(* IEC 61131-3 sources: PID/Source/IMM/ieccontrol/Ejector1, 4 files *)

(* ---- FBInsteadIOConfig.pu ---- *)
FUNCTION_BLOCK FBInsteadIOConfig #DUMMY_EDIT_BLOCK

VAR_INPUT
 IOPath : STRING(255);
END_VAR

VAR
 SystemPath : STRING(255) := '/harddisk0/application/control/config/KeStudio_generated/Device1/PlcIo.cfgr';
END_VAR
#BEGIN_EDIT_BLOCK
Stable_Copy := KFILE_Copy(IOPath,SystemPath);

;#END_EDIT_BLOCK END_FUNCTION_BLOCK

#END_OF_IEC_PART

@Puma @IecEditor 6 152 @Pou 25
@@@BEG_Comment@@@

@@@END_Comment@@@

@BEG_Contents

@BEG_Func
@RT(17)FuncTreeContainer
0
@END_Func

@BEG_Const
@RT(18)ConstTreeContainer
0
@END_Const

@BEG_Export

@BEG_Kind
@FUNCTION_BLOCK @RT(17)FBInsteadIOConfig @STRUCTURED_TEXT
@RT(0) @RT(0) @RT(0)
@END_Kind

@BEG_Dcl
@RT(16)DclTreeContainer
2
@Var @RT(10)SystemPath @RT(0) @T @F @DT @RT(11)STRING(255) @RT(0) @T @T @STRING 0 @F @RT(3)255 @F
@F @F
@T
@BEG_Attrib
3 @RT(77)'/harddisk0/application/control/config/KeStudio_generated/Device1/PlcIo.cfgr' @RT(0) @RT(0)
@END_Attrib
1 0 @F @F @F @F

@Var @RT(6)IOPath @RT(0) @T @F @DT @RT(11)STRING(255) @RT(0) @T @T @STRING 0 @F @RT(3)255 @F
@F @F
@T
@BEG_Attrib
3 @RT(0) @RT(0) @RT(0)
@END_Attrib
1 1 @F @F @F @F

@END_Dcl

@END_Export

@BEG_Body
@TL(2)
Stable_Copy := KFILE_Copy(IOPath,SystemPath);

@END_Body

@END_Contents

(* ---- FBReadIOConfigFiles.pu ---- *)
IMPORT_OVER_LISTFILE
 KFILE_Status
, UsbFilesArray

END_IMPORT

FUNCTION_BLOCK FBReadIOConfigFiles #DUMMY_EDIT_BLOCK

VAR_INPUT
 PLCFiles : STRING(255) := '/harddisk0/PLCIO';
END_VAR

VAR_OUTPUT
 PathArray : UsbFilesArray;
END_VAR

VAR_TEMP
 j : DINT;
END_VAR

VAR
 Stable_Free : KFILE_Status;
 Stable_First : KFILE_Status;
 Stable_Next : KFILE_Status;
 i : LINT;
 harddisk0 : STRING(255) := '/harddisk0';
 s : STRING(255);
 s2 : STRING(255);
END_VAR

(* IecGraph-Code *)

(* init step *)
INITIAL_STEP Step1:
Action1 (P);
END_STEP

ACTION Action1: #BEGIN_EDIT_BLOCK
//Check harddisk left memory
Stable_Free :=  KFILE_VolumeFree(harddisk0,i)

;#END_EDIT_BLOCK END_ACTION (*Action1*)

(* steps *)
STEP Step4:
Action3 (P);
END_STEP

ACTION Action3: #BEGIN_EDIT_BLOCK
//get first file name in the file
Stable_First := KFILE_GetFirst(PLCFiles,s);
PathArray[1] := s;
s2 := s;
FOR j :=2 TO 10 DO
   //get other file name in the file
   Stable_Next := KFILE_GetNext(s2,s2);
   PathArray[j] := s2;
END_FOR;
//Now all file name in sv_PathArray

;#END_EDIT_BLOCK END_ACTION (*Action3*)
STEP Step2:
Action5 (N);
END_STEP

ACTION Action5: #BEGIN_EDIT_BLOCK
RETURN;

;#END_EDIT_BLOCK END_ACTION (*Action5*)

(* transitions *)
TRANSITION Trans3 (* Trans3 *) FROM Step1 TO Step4 :=  #BEGIN_EDIT_BLOCK
Stable_Free = KFILE_Status_OK
;#END_EDIT_BLOCK
END_TRANSITION

TRANSITION Trans5 (* Trans5 *) FROM Step4 TO Step2 :=  #BEGIN_EDIT_BLOCK
Stable_Next = KFILE_Status_NOTOK
;#END_EDIT_BLOCK
END_TRANSITION

TRANSITION Trans2 (* Trans2 *) FROM Step2 TO Step1 :=  #BEGIN_EDIT_BLOCK
TRUE
;#END_EDIT_BLOCK
END_TRANSITION

(* end IecGraph-Code *)
(* sfc-code *)
(* end sfc-code *)

END_FUNCTION_BLOCK

#END_OF_IEC_PART

@Puma @IecEditor 6 152 @Pou 25
@@@BEG_Comment@@@

@@@END_Comment@@@

@BEG_Contents

@BEG_Func
@RT(17)FuncTreeContainer
0
@END_Func

@BEG_Const
@RT(18)ConstTreeContainer
0
@END_Const

@BEG_Export

@BEG_Kind
@FUNCTION_BLOCK @RT(19)FBReadIOConfigFiles @SEQUENTIAL_FLOW_CHART
@RT(0) @RT(0) @RT(0)
@END_Kind

@BEG_Dcl
@RT(16)DclTreeContainer
10
@Var @RT(11)Stable_Free @RT(0) @T @T @DERIVED 0 @T @T @DT @RT(12)KFILE_Status @RT(0) @T @T @UNKNOWN 0 @F
@F @F
@T
@BEG_Attrib
3 @RT(0) @RT(0) @RT(0)
@END_Attrib
1 0 @F @F @F @F

@Var @RT(12)Stable_First @RT(0) @T @T @DERIVED 0 @T @T @DT @RT(12)KFILE_Status @RT(0) @T @T @UNKNOWN 0 @F
@F @F
@T
@BEG_Attrib
3 @RT(0) @RT(0) @RT(0)
@END_Attrib
1 0 @F @F @F @F

@Var @RT(11)Stable_Next @RT(0) @T @T @DERIVED 0 @T @T @DT @RT(12)KFILE_Status @RT(0) @T @T @UNKNOWN 0 @F
@F @F
@T
@BEG_Attrib
3 @RT(0) @RT(0) @RT(0)
@END_Attrib
1 0 @F @F @F @F

@Var @RT(1)i @RT(0) @T @F @DT @RT(4)LINT @RT(0) @T @T @BASIC 0 @F
@F @F
@T
@BEG_Attrib
3 @RT(0) @RT(0) @RT(0)
@END_Attrib
1 0 @F @F @F @F

@Var @RT(1)j @RT(0) @T @F @DT @RT(4)DINT @RT(0) @T @T @BASIC 0 @F
@F @F
@T
@BEG_Attrib
3 @RT(0) @RT(0) @RT(0)
@END_Attrib
1 4 @F @F @F @F

@Var @RT(9)harddisk0 @RT(0) @T @F @DT @RT(11)STRING(255) @RT(0) @T @T @STRING 0 @F @RT(3)255 @F
@F @F
@T
@BEG_Attrib
3 @RT(12)'/harddisk0' @RT(0) @RT(0)
@END_Attrib
1 0 @F @F @F @F

@Var @RT(8)PLCFiles @RT(0) @T @F @DT @RT(11)STRING(255) @RT(0) @T @T @STRING 0 @F @RT(3)255 @F
@F @F
@T
@BEG_Attrib
3 @RT(18)'/harddisk0/PLCIO' @RT(0) @RT(0)
@END_Attrib
1 1 @F @F @F @F

@Var @RT(9)PathArray @RT(0) @T @T @DERIVED 0 @F @RT(13)UsbFilesArray @F
@T
@BEG_Attrib
3 @RT(0) @RT(0) @RT(0)
@END_Attrib
1 3 @F @F @F @F

@Var @RT(1)s @RT(0) @T @F @DT @RT(11)STRING(255) @RT(0) @T @T @STRING 0 @F @RT(3)255 @F
@F @F
@T
@BEG_Attrib
3 @RT(0) @RT(0) @RT(0)
@END_Attrib
1 0 @F @F @F @F

@Var @RT(2)s2 @RT(0) @T @F @DT @RT(11)STRING(255) @RT(0) @T @T @STRING 0 @F @RT(3)255 @F
@F @F
@T
@BEG_Attrib
3 @RT(0) @RT(0) @RT(0)
@END_Attrib
1 0 @F @F @F @F

@END_Dcl

@END_Export

@BEG_SfcBody
2 2 2

@BEG_SfcData 2
@StepSeq @RT(4)sseq @F 1
@Loop @RT(4)loop @F 2
@StepSeq @RT(3)seq @F 5
@Step @RT(5)Step1 @F @T @F @F @RT(0) @F
@AcbCont @RT(7)unnamed @F 1
@Acb @RT(7)Action1 @F @T @RT(1)P @RT(0) @F @F @T @TL(3)
//Check harddisk left memory
Stable_Free :=  KFILE_VolumeFree(harddisk0,i)

@F

@Trans @RT(6)Trans3 @F @T @F @F @T @T @TL(2)
Stable_Free = KFILE_Status_OK

@RT(6)Trans3 @F
@Step @RT(5)Step4 @F @F @F @F @RT(0) @F
@AcbCont @RT(7)unnamed @F 1
@Acb @RT(7)Action3 @F @T @RT(1)P @RT(0) @F @F @T @TL(11)
//get first file name in the file
Stable_First := KFILE_GetFirst(PLCFiles,s);
PathArray[1] := s;
s2 := s;
FOR j :=2 TO 10 DO
   //get other file name in the file
   Stable_Next := KFILE_GetNext(s2,s2);
   PathArray[j] := s2;
END_FOR;
//Now all file name in sv_PathArray

@F

@Trans @RT(6)Trans5 @F @T @F @F @T @T @TL(2)
Stable_Next = KFILE_Status_NOTOK

@RT(6)Trans5 @F
@Step @RT(5)Step2 @F @F @F @F @RT(0) @F
@AcbCont @RT(7)unnamed @F 1
@Acb @RT(7)Action5 @F @T @RT(1)N @RT(0) @F @F @T @TL(2)
RETURN;

@F

@Trans @RT(6)Trans2 @F @T @T @T @T @T @TL(2)
TRUE

@RT(6)Trans2 @F

@END_SfcData
@SaActions 0
@SaTrans 0
@SaExits 0
@END_SfcBody

@END_Contents

(* ---- ABMeasure.pu ---- *)
IMPORT_OVER_LISTFILE
 GET_MY_FU_NAME
, KSWO_AddVariable
, WRITE_SVREAL_DIRECT
, FAddToScopeGroup
, START_PROCESS_ALGORITHM
, STOP_PROCESS_ALGORITHM
, KFILE_VolumeFree
, KFILE_GetNext
, KFILE_GetFirst
, KAPPL_LintabData
, KAPPL_MeasureMonitoring
, UsbFilesArray
//  UsbFile
, FBReadIOConfigFiles
, KSWO_Status
, ABMeasureAI
, TON
, KFILE_Status
, ABPID

END_IMPORT

ALGORITHM_BLOCK ABMeasure #DUMMY_EDIT_BLOCK

SYSTEM_VAR
 sv_rEjectorPosition : REAL;
 sv_EjectorLintab : KAPPL_LintabData;
 ai_Position : REAL;
 sv_bTransducerError : BOOL;
 sv_bDeviceReady : BOOL;
 sv_rEjectorVelocity : REAL;
 sv_EjectorMonitorMeas : KAPPL_MeasureMonitoring;
 sv_Ek : REAL;
 sv_Ek_1 : REAL;
 sv_Ek_2 : REAL;
 sv_Uk : REAL;
 sv_Ui : REAL;
 sv_Uk_1 : REAL;
 sv_Uk_2 : REAL;
 sv_Uk_3 : REAL;
 di_ButtonBwd : BOOL (* Panelbutton *);
 di_ButtonFwd : BOOL (* Panelbutton *);
 ao_pid : REAL;
 sv_PathArray : UsbFilesArray;
 // sv_PathDisplay : UsbFile;
 sv_rActOutput : INT;
 sv_rSetOutput : INT;
 sv_bStartPID : BOOL;
END_VAR

SYSTEM_OBJECT
 TaskAnalog : TASK;
 TaskSlow : TASK;
 PU_Task_7 : TASK;
 // erCopyDone : ALARM;
END_OBJECT

VAR
 t : REAL := 0.2;
 T : REAL;
 Kp : REAL := 0.05;
 Ti : REAL;
 ti : REAL := 0.05;
 Td : REAL;
 td : REAL := 2.0;
 A : REAL;
 B : REAL;
 C : REAL;
 ai_pid : REAL := 10.0;
 PWMPeriod : TIME;
 T_PID : REAL;
 L_T : REAL;
 H_T : REAL;
 DutyRatio : REAL;
 fbReadIOConfigFiles : FBReadIOConfigFiles;
END_VAR

PROCESS_ALGORITHM paInitDebugMeasurement ON TaskSlow AUTOSTART

VAR
 fuName : STRING(255);
 variableName : STRING(255);
 swoState : KSWO_Status;
 b : BOOL;
END_VAR
#BEGIN_EDIT_BLOCK
fuName := GET_MY_FU_NAME();
variableName := CONCAT(fuName,'.rPosition mm');
swoState := KSWO_AddVariable( Task := TaskAnalog,
                              Name := variableName,
                              Variable := sv_rEjectorPosition);
b := FAddToScopeGroup(Task := TaskAnalog,
                      Name := variableName,
                      GroupId := cScopeGroupEjector);
variableName := CONCAT(fuName,'.rVelocity mm/s');
swoState := KSWO_AddVariable( Task := TaskAnalog,
                              Name := variableName,
                              Variable := sv_rEjectorVelocity);
b := FAddToScopeGroup(Task := TaskAnalog,
                      Name := variableName,
                      GroupId := cScopeGroupEjector);

    variableName := CONCAT(fuName,'.sv_Ek');
swoState := KSWO_AddVariable( Task := TaskAnalog,
                              Name := variableName,
                              Variable := sv_Ek);

    variableName := CONCAT(fuName,'.sv_Uk');
swoState := KSWO_AddVariable( Task := TaskAnalog,
                              Name := variableName,
                              Variable := sv_Uk);

    variableName := CONCAT(fuName,'.sv_Ui');
swoState := KSWO_AddVariable( Task := TaskAnalog,
                              Name := variableName,
                              Variable := sv_Ui);

    variableName := CONCAT(fuName,'.ao_pid');
swoState := KSWO_AddVariable( Task := TaskAnalog,
                              Name := variableName,
                              Variable := ao_pid);

    variableName := CONCAT(fuName,'.ai_pid');
swoState := KSWO_AddVariable( Task := TaskAnalog,
                              Name := variableName,
                              Variable := ai_pid);

    variableName := CONCAT(fuName,'.sv_rActOutput');
swoState := KSWO_AddVariable( Task := TaskAnalog,
                              Name := variableName,
                              Variable := sv_rActOutput);
    variableName := CONCAT(fuName,'.sv_rSetOutput');
swoState := KSWO_AddVariable( Task := TaskAnalog,
                              Name := variableName,
                              Variable := sv_rSetOutput);

STOP_PROCESS_ALGORITHM();

;#END_EDIT_BLOCK END_ALGORITHM

PROCESS_ALGORITHM paMeasure ON TaskAnalog AUTOSTART

VAR_TEMP
 b : BOOL;
END_VAR

VAR
 abEjectorMeasure : ABMeasureAI;
END_VAR

(* IecGraph-Code *)

(* init step *)
INITIAL_STEP S_Start:
END_STEP

(* steps *)
STEP S_Stop:
AStop (P);
END_STEP

ACTION AStop: #BEGIN_EDIT_BLOCK
STOP_PROCESS_ALGORITHM();

;#END_EDIT_BLOCK END_ACTION (*AStop*)
STEP S_Init:
AInitMeasureBlock (P);
END_STEP

STEP S_Measure:
AMeasure (N);
END_STEP

(* transitions *)
TRANSITION TLinked (* TLinked *) FROM S_Start TO S_Init :=  #BEGIN_EDIT_BLOCK
IS_LINKED(ai_Position)
;#END_EDIT_BLOCK
END_TRANSITION

TRANSITION TNotLinked (* TNotLinked *) FROM S_Start TO S_Stop :=  #BEGIN_EDIT_BLOCK
NOT IS_LINKED(ai_Position)
;#END_EDIT_BLOCK
END_TRANSITION

TRANSITION TStop (* TStop *) FROM S_Stop TO S_Start :=  #BEGIN_EDIT_BLOCK
TRUE
;#END_EDIT_BLOCK
END_TRANSITION

TRANSITION TInitDone (* TInitDone *) FROM S_Init TO S_Measure :=  #BEGIN_EDIT_BLOCK
TRUE
;#END_EDIT_BLOCK
END_TRANSITION

(* end IecGraph-Code *)
(* sfc-code *)

(* stand alone actions *)
ACTION AMeasure: #BEGIN_EDIT_BLOCK

abEjectorMeasure.aRun(bIdle := sv_bDeviceReady);
sv_bTransducerError := abEjectorMeasure.aRun.bSensorError;
b := WRITE_SVREAL_DIRECT(sv_rEjectorPosition, abEjectorMeasure.aRun.rValue);
b := WRITE_SVREAL_DIRECT(sv_rEjectorVelocity, abEjectorMeasure.aRun.rVelocity);

;#END_EDIT_BLOCK END_ACTION (*AMeasure*)
ACTION AInitMeasureBlock: #BEGIN_EDIT_BLOCK

abEjectorMeasure.aInit(sRawValue := 'Ejector1.ai_Position',
                        pLintab := @sv_EjectorLintab);

abEjectorMeasure.aInitMonitoring(bEnable := sv_EjectorMonitorMeas.EnableMonitoring,
                                 rLowLimit := sv_EjectorMonitorMeas.LowerLimit,
                                 bLimitation := sv_EjectorMonitorMeas.Limitation,
                                 rFailureFactor := sv_EjectorMonitorMeas.FailureFactor);

;#END_EDIT_BLOCK END_ACTION (*AInitMeasureBlock*)
(* end sfc-code *)

END_ALGORITHM

PROCESS_ALGORITHM paPID ON TaskAnalog

(* IecGraph-Code *)

(* init step *)
INITIAL_STEP Step1:
Action223 (P);
END_STEP

ACTION Action223: #BEGIN_EDIT_BLOCK
ai_pid := 10.0;
t := 0.1;
td := 2.0;
ti := 0.05;
Kp := 0.2;

;#END_EDIT_BLOCK END_ACTION (*Action223*)

(* steps *)
STEP Step2:
Action2 (P);
END_STEP

ACTION Action2: #BEGIN_EDIT_BLOCK
sv_Ek := 0.0;
sv_Ek_1 := 0.0;
sv_Ek_2 := 0.0;
sv_Uk := 0.0;
sv_Uk_1 := 0.0;
sv_Uk_2 := 0.0;
sv_Uk_3 := 0.0;

;#END_EDIT_BLOCK END_ACTION (*Action2*)
STEP Step4:
END_STEP

STEP Step3:
Action3 (P);
END_STEP

ACTION Action3: #BEGIN_EDIT_BLOCK
T := 1.0/t;
Td := 1.0/td;
Ti := 1.0/ti;
A := Kp*(1.0 + T/Ti + Td/T);
B := Kp*(1.0 + 2.0*Td/T);
C := Kp*Td/T;
sv_Uk_3 := sv_Uk_2;
sv_Uk_2 := sv_Uk_1;
sv_Uk_1 := sv_Uk;
sv_Ek_2 := sv_Ek_1;
sv_Ek_1 := sv_Ek;
sv_Ek := ai_pid - sv_Uk;
sv_Ui := A*sv_Ek + B*sv_Ek_1 + C*sv_Ek_2;
ao_pid := sv_Uk_1 + sv_Ui;
sv_Uk := sv_Uk_1 + sv_Ui;

;#END_EDIT_BLOCK END_ACTION (*Action3*)

(* transitions *)
GO_ON_TRANSITION Trans1 (* Trans1 *) FROM Step1 TO Step2 :=  #BEGIN_EDIT_BLOCK
TRUE
;#END_EDIT_BLOCK
END_TRANSITION

TRANSITION Trans4 (* Trans4 *) FROM Step2 TO Step4 :=  #BEGIN_EDIT_BLOCK
TRUE
;#END_EDIT_BLOCK
END_TRANSITION

TRANSITION Trans2 (* Trans2 *) FROM Step4 TO Step3 :=  #BEGIN_EDIT_BLOCK
Step4.T > t#0.1s
;#END_EDIT_BLOCK
END_TRANSITION

GO_ON_TRANSITION Trans5 (* Trans5 *) FROM Step3 TO Step4 :=  #BEGIN_EDIT_BLOCK
TRUE
;#END_EDIT_BLOCK
END_TRANSITION

(* end IecGraph-Code *)
(* sfc-code *)
(* end sfc-code *)

END_ALGORITHM

POSTUPDATE_ALGORITHM p ON PU_Task_7 WITH di_ButtonBwd,di_ButtonFwd

VAR
 a : INT;
END_VAR
#BEGIN_EDIT_BLOCK

IF di_ButtonFwd THEN
   START_PROCESS_ALGORITHM(paPID);
   START_PROCESS_ALGORITHM(paPWM);

END_IF;

IF di_ButtonBwd THEN
   STOP_PROCESS_ALGORITHM(paPID);
   STOP_PROCESS_ALGORITHM(paPWM);
END_IF;
//year=(year%100==0)?(year%400==0?1:0):(year%4==0?1:0)

;#END_EDIT_BLOCK END_ALGORITHM

PROCESS_ALGORITHM paPWM ON TaskAnalog

VAR
 fbTON : TON;
 do : BOOL;
END_VAR

(* IecGraph-Code *)

(* init step *)
INITIAL_STEP Step1:
Action20 (P);
END_STEP

ACTION Action20: #BEGIN_EDIT_BLOCK
PWMPeriod := t#2s;

;#END_EDIT_BLOCK END_ACTION (*Action20*)

(* steps *)
STEP Step2:
Action2 (P);
END_STEP

ACTION Action2: #BEGIN_EDIT_BLOCK
T_PID := ao_pid;
L_T := 8.0;
H_T := 10.0;
IF T_PID < L_T THEN
   DutyRatio := 1.0;
ELSE IF T_PID >= H_T - 0.1 THEN
   DutyRatio := 0.0;
ELSE
   DutyRatio := (T_PID - L_T) /(H_T - L_T);
END_IF;
END_IF;
fbTON(IN := FALSE);

;#END_EDIT_BLOCK END_ACTION (*Action2*)
STEP Step5:
Action3 (N);
END_STEP

ACTION Action3: #BEGIN_EDIT_BLOCK
fbTON(IN := TRUE,
     // PT := REAL_TO_TIME(TIME_TO_REAL(PWMPeriod) * DutyRatio);
            PT := PWMPeriod * DutyRatio);
IF fbTON.Q THEN
   do := FALSE;
ELSE
   do := TRUE;
END_IF;

;#END_EDIT_BLOCK END_ACTION (*Action3*)
STEP Step3:
END_STEP

(* transitions *)
TRANSITION Trans1 (* Trans1 *) FROM Step1 TO Step2 :=  #BEGIN_EDIT_BLOCK
TRUE
;#END_EDIT_BLOCK
END_TRANSITION

TRANSITION Trans2 (* Trans2 *) FROM Step2 TO Step5 :=  #BEGIN_EDIT_BLOCK
TRUE
;#END_EDIT_BLOCK
END_TRANSITION

TRANSITION Trans11 (* Trans11 *) FROM Step5 TO Step3 :=  #BEGIN_EDIT_BLOCK
Step5.T > PWMPeriod
;#END_EDIT_BLOCK
END_TRANSITION

TRANSITION Trans12 (* Trans12 *) FROM Step3 TO Step2 :=  #BEGIN_EDIT_BLOCK
TRUE
;#END_EDIT_BLOCK
END_TRANSITION

(* end IecGraph-Code *)
(* sfc-code *)
(* end sfc-code *)

END_ALGORITHM

POSTUPDATE_ALGORITHM USB ON PU_Task_7 WITH di_ButtonBwd,di_ButtonFwd

VAR
 PLCFiles : STRING(255) := '/harddisk0/PLCIO';
END_VAR
#BEGIN_EDIT_BLOCK
IF di_ButtonBwd THEN
   START_PROCESS_ALGORITHM(paUSB);
END_IF;
IF di_ButtonFwd THEN
   STOP_PROCESS_ALGORITHM(paUSB);
END_IF;

;#END_EDIT_BLOCK END_ALGORITHM

PROCESS_ALGORITHM paUSB ON TaskAnalog

VAR_TEMP
 j : DINT;
END_VAR

VAR
 Stable_Free : KFILE_Status;
 Stable_Delete : KFILE_Status;
 Stable_Copy : KFILE_Status;
 Stable_Next : KFILE_Status;
 Stable_First : KFILE_Status;
 Stable_Copy2 : KFILE_Status;
 Stable_Rename : KFILE_Status;
 i : LINT;
 SystemPath : STRING(255) := '/harddisk0/application/control/config/KeStudio_generated/Device1/PlcIo.cfgr';
 s : STRING(255);
 s2 : STRING(255);
 harddisk0 : STRING(255) := '/harddisk0';
 PLCFiles : STRING(255) := '/harddisk0';
END_VAR

(* IecGraph-Code *)

(* init step *)
INITIAL_STEP Step1:
Action1 (P);
END_STEP

ACTION Action1: #BEGIN_EDIT_BLOCK
//Check harddisk left memory
Stable_Free :=  KFILE_VolumeFree(harddisk0,i)

;#END_EDIT_BLOCK END_ACTION (*Action1*)

(* steps *)
STEP Step4:
Action3 (P);
END_STEP

ACTION Action3: #BEGIN_EDIT_BLOCK
//get first file name in the file
Stable_First := KFILE_GetFirst(PLCFiles,s);
sv_PathArray[1] := s;
s2 := s;
FOR j :=2 TO 10 DO
   //get other file name in the file
   Stable_Next := KFILE_GetNext(s2,s2);
   sv_PathArray[j] := s2;
END_FOR;
//Now all file name in sv_PathArray

;#END_EDIT_BLOCK END_ACTION (*Action3*)
STEP Step2:
Action5 (N);
END_STEP

ACTION Action5: #BEGIN_EDIT_BLOCK

STOP_PROCESS_ALGORITHM();

;#END_EDIT_BLOCK END_ACTION (*Action5*)

(* transitions *)
TRANSITION Trans3 (* Trans3 *) FROM Step1 TO Step4 :=  #BEGIN_EDIT_BLOCK
Stable_Free = KFILE_Status_OK
;#END_EDIT_BLOCK
END_TRANSITION

TRANSITION Trans5 (* Trans5 *) FROM Step4 TO Step2 :=  #BEGIN_EDIT_BLOCK
Stable_Next = KFILE_Status_NOTOK
;#END_EDIT_BLOCK
END_TRANSITION

TRANSITION Trans2 (* Trans2 *) FROM Step2 TO Step1 :=  #BEGIN_EDIT_BLOCK
TRUE
;#END_EDIT_BLOCK
END_TRANSITION

(* end IecGraph-Code *)
(* sfc-code *)
(* end sfc-code *)

END_ALGORITHM

// POSTUPDATE_ALGORITHM pchoose ON PU_Task_7 WITH sv_bUse1,sv_bUse2,sv_bUse3,sv_bUse4,sv_bUse5,sv_bUse6,sv_bUse7,sv_bUse8,sv_bUse9,sv_bUse10

// VAR
 // Stable_Copy : KFILE_Status;
 // SystemPath : STRING(255) := '/harddisk0/application/control/config/KeStudio_generated/Device1/PlcIo.cfgr';
// END_VAR
// #BEGIN_EDIT_BLOCK
// IF sv_bUse1 THEN
// Stable_Copy := KFILE_Copy(sv_PathDisplay.plc1,SystemPath);
// END_IF;
//
// IF sv_bUse2 THEN
// Stable_Copy := KFILE_Copy(sv_PathDisplay.plc2,SystemPath);
// END_IF;
//
// IF sv_bUse3  THEN
// Stable_Copy := KFILE_Copy(sv_PathDisplay.plc3,SystemPath);
// END_IF;
//
// IF sv_bUse4 THEN
// Stable_Copy := KFILE_Copy(sv_PathDisplay.plc4,SystemPath);
// END_IF;
//
// IF sv_bUse5 THEN
// Stable_Copy := KFILE_Copy(sv_PathDisplay.plc5,SystemPath);
// END_IF;
//
// IF sv_bUse6 THEN
// Stable_Copy := KFILE_Copy(sv_PathDisplay.plc6,SystemPath);
// END_IF;
//
// IF sv_bUse7 THEN
// Stable_Copy := KFILE_Copy(sv_PathDisplay.plc7,SystemPath);
// END_IF;
//
// IF sv_bUse8 THEN
// Stable_Copy := KFILE_Copy(sv_PathDisplay.plc8,SystemPath);
// END_IF;
//
// IF sv_bUse9 THEN
// Stable_Copy := KFILE_Copy(sv_PathDisplay.plc9,SystemPath);
// END_IF;
//
// IF sv_bUse10 THEN
// Stable_Copy := KFILE_Copy(sv_PathDisplay.plc10,SystemPath);
// END_IF;
//

// ;#END_EDIT_BLOCK END_ALGORITHM

// PROCESS_ALGORITHM paPIDCalc ON TaskAnalog AUTOSTART

// #BEGIN_EDIT_BLOCK
// Td := 1.0/td;
// Ti := 1.0/ti;
// A := Kp*(1.0 + T/Ti + Td/T);
// B := Kp*(1.0 + 2.0*Td/T);
// C := Kp*Td/T;
// sv_Uk_3 := sv_Uk_2;
// sv_Uk_2 := sv_Uk_1;
// sv_Uk_1 := sv_Uk;
// sv_Ek_2 := sv_Ek_1;
// sv_Ek_1 := sv_Ek;
// sv_Ek := ai_pid - sv_Uk;
// sv_Ui := A*sv_Ek + B*sv_Ek_1 + C*sv_Ek_2;
// ao_pid := sv_Uk_1 + sv_Ui;
// sv_Uk := sv_Uk_1 + sv_Ui;

// ;#END_EDIT_BLOCK END_ALGORITHM

PROCESS_ALGORITHM pStaratPID ON TaskSlow AUTOSTART

VAR
 iKp : INT := 2;
 iKd : INT := 1;
 iKi : INT := 1;
 iFilter : INT := 1023;
 iIntegr : INT := 0;
 abPID : ABPID;
END_VAR
#BEGIN_EDIT_BLOCK
IF sv_bStartPID THEN
    abPID.aPID(iAct := (sv_rActOutput * 32/ 100),
         iSet := (sv_rSetOutput * 32 / 100),
         iKp := iKp,
         iKi := iKi,
         iKd := iKd,
         iC0 := iFilter,
         iYlow := -32,
         iYup := 32,
         iIntegr := iIntegr,
         iY => sv_rActOutput);
   iIntegr := abPID.aPID.iIntegr;

END_IF;

;#END_EDIT_BLOCK END_ALGORITHM

END_ALGORITHM_BLOCK

#END_OF_IEC_PART

@Puma @IecEditor 6 103 @Pou 25
@@@BEG_Comment@@@

@@@END_Comment@@@

@BEG_Contents

@BEG_Func
@RT(17)FuncTreeContainer
9
@Var @RT(14)GET_MY_FU_NAME @RT(0) @T @T @DERIVED 0 @F @RT(22)KEBA_STANDARD_FUNCTION @F
@T
@BEG_Attrib
0 @RT(0) @RT(0)
@END_Attrib
1 1 @F @F @F @F

@Var @RT(16)KSWO_AddVariable @RT(0) @T @T @DERIVED 0 @F @RT(22)KEBA_STANDARD_FUNCTION @F
@T
@BEG_Attrib
0 @RT(0) @RT(0)
@END_Attrib
1 1 @F @F @F @F

@Var @RT(19)WRITE_SVREAL_DIRECT @RT(0) @T @T @DERIVED 0 @F @RT(22)KEBA_STANDARD_FUNCTION @F
@T
@BEG_Attrib
0 @RT(0) @RT(0)
@END_Attrib
1 1 @F @F @F @F

@Var @RT(16)FAddToScopeGroup @RT(0) @T @T @DERIVED 0 @F @RT(8)FUNCTION @F
@T
@BEG_Attrib
0 @RT(0) @RT(0)
@END_Attrib
1 1 @F @F @F @F

@Var @RT(23)START_PROCESS_ALGORITHM @RT(0) @T @T @DERIVED 0 @F @RT(23)KEBA_STANDARD_PROCEDURE @F
@T
@BEG_Attrib
0 @RT(0) @RT(0)
@END_Attrib
1 1 @F @F @F @F

@Var @RT(22)STOP_PROCESS_ALGORITHM @RT(0) @T @T @DERIVED 0 @F @RT(23)KEBA_STANDARD_PROCEDURE @F
@T
@BEG_Attrib
0 @RT(0) @RT(0)
@END_Attrib
1 1 @F @F @F @F

@Var @RT(16)KFILE_VolumeFree @RT(0) @T @T @DERIVED 0 @F @RT(22)KEBA_STANDARD_FUNCTION @F
@T
@BEG_Attrib
0 @RT(0) @RT(0)
@END_Attrib
1 1 @F @F @F @F

@Var @RT(13)KFILE_GetNext @RT(0) @T @T @DERIVED 0 @F @RT(22)KEBA_STANDARD_FUNCTION @F
@T
@BEG_Attrib
0 @RT(0) @RT(0)
@END_Attrib
1 1 @F @F @F @F

@Var @RT(14)KFILE_GetFirst @RT(0) @T @T @DERIVED 0 @F @RT(22)KEBA_STANDARD_FUNCTION @F
@T
@BEG_Attrib
0 @RT(0) @RT(0)
@END_Attrib
1 1 @F @F @F @F

@END_Func

@BEG_Const
@RT(18)ConstTreeContainer
0
@END_Const

@BEG_Export

@BEG_Kind
@ALGORITHM_BLOCK @RT(9)ABMeasure @STRUCTURED_TEXT
@RT(0) @RT(0) @RT(0)
@END_Kind

@BEG_Dcl
@RT(16)DclTreeContainer
44
@Var @RT(19)sv_rEjectorPosition @RT(0) @T @F @DT @RT(4)REAL @RT(0) @T @T @BASIC 0 @F
@F @F
@T
@BEG_Attrib
3 @RT(0) @RT(0) @RT(0)
@END_Attrib
1 8 @F @F @F @F

@Var @RT(16)sv_EjectorLintab @RT(0) @T @T @DERIVED 0 @T @T @DT @RT(16)KAPPL_LintabData @RT(0) @T @T @UNKNOWN 0 @F
@F @F
@T
@BEG_Attrib
3 @RT(0) @RT(0) @RT(0)
@END_Attrib
1 8 @F @F @F @F

@Var @RT(11)ai_Position @RT(0) @T @F @DT @RT(4)REAL @RT(0) @T @T @BASIC 0 @F
@F @F
@T
@BEG_Attrib
3 @RT(0) @RT(0) @RT(0)
@END_Attrib
1 8 @F @F @F @F

@Var @RT(19)sv_bTransducerError @RT(0) @T @F @DT @RT(4)BOOL @RT(0) @T @T @BASIC 0 @F
@F @F
@T
@BEG_Attrib
3 @RT(0) @RT(0) @RT(0)
@END_Attrib
1 8 @F @F @F @F

@Var @RT(15)sv_bDeviceReady @RT(0) @T @F @DT @RT(4)BOOL @RT(0) @T @T @BASIC 0 @F
@F @F
@T
@BEG_Attrib
3 @RT(0) @RT(0) @RT(0)
@END_Attrib
1 8 @F @F @F @F

@Var @RT(19)sv_rEjectorVelocity @RT(0) @T @F @DT @RT(4)REAL @RT(0) @T @T @BASIC 0 @F
@F @F
@T
@BEG_Attrib
3 @RT(0) @RT(0) @RT(0)
@END_Attrib
1 8 @F @F @F @F

@Var @RT(21)sv_EjectorMonitorMeas @RT(0) @T @T @DERIVED 0 @T @T @DT @RT(23)KAPPL_MeasureMonitoring @RT(0) @T @T @UNKNOWN 0 @F
@F @F
@T
@BEG_Attrib
3 @RT(0) @RT(0) @RT(0)
@END_Attrib
1 8 @F @F @F @F

@Var @RT(10)TaskAnalog @RT(0) @T @F @DT @RT(4)TASK @RT(0) @T @T @BASIC 0 @F
@F @F
@T
@BEG_Attrib
3 @RT(0) @RT(0) @RT(0)
@END_Attrib
1 7 @F @F @F @F

@Var @RT(8)TaskSlow @RT(0) @T @F @DT @RT(4)TASK @RT(0) @T @T @BASIC 0 @F
@F @F
@T
@BEG_Attrib
3 @RT(0) @RT(0) @RT(0)
@END_Attrib
1 7 @F @F @F @F

@Var @RT(5)sv_Ek @RT(0) @T @F @DT @RT(4)REAL @RT(0) @T @T @BASIC 0 @F
@F @F
@T
@BEG_Attrib
3 @RT(0) @RT(0) @RT(0)
@END_Attrib
1 8 @F @F @F @F

@Var @RT(7)sv_Ek_1 @RT(0) @T @F @DT @RT(4)REAL @RT(0) @T @T @BASIC 0 @F
@F @F
@T
@BEG_Attrib
3 @RT(0) @RT(0) @RT(0)
@END_Attrib
1 8 @F @F @F @F

@Var @RT(7)sv_Ek_2 @RT(0) @T @F @DT @RT(4)REAL @RT(0) @T @T @BASIC 0 @F
@F @F
@T
@BEG_Attrib
3 @RT(0) @RT(0) @RT(0)
@END_Attrib
1 8 @F @F @F @F

@Var @RT(5)sv_Uk @RT(0) @T @F @DT @RT(4)REAL @RT(0) @T @T @BASIC 0 @F
@F @F
@T
@BEG_Attrib
3 @RT(0) @RT(0) @RT(0)
@END_Attrib
1 8 @F @F @F @F

@Var @RT(5)sv_Ui @RT(0) @T @F @DT @RT(4)REAL @RT(0) @T @T @BASIC 0 @F
@F @F
@T
@BEG_Attrib
3 @RT(0) @RT(0) @RT(0)
@END_Attrib
1 8 @F @F @F @F

@Var @RT(7)sv_Uk_1 @RT(0) @T @F @DT @RT(4)REAL @RT(0) @T @T @BASIC 0 @F
@F @F
@T
@BEG_Attrib
3 @RT(0) @RT(0) @RT(0)
@END_Attrib
1 8 @F @F @F @F

@Var @RT(7)sv_Uk_2 @RT(0) @T @F @DT @RT(4)REAL @RT(0) @T @T @BASIC 0 @F
@F @F
@T
@BEG_Attrib
3 @RT(0) @RT(0) @RT(0)
@END_Attrib
1 8 @F @F @F @F

@Var @RT(7)sv_Uk_3 @RT(0) @T @F @DT @RT(4)REAL @RT(0) @T @T @BASIC 0 @F
@F @F
@T
@BEG_Attrib
3 @RT(0) @RT(0) @RT(0)
@END_Attrib
1 8 @F @F @F @F

@Var @RT(1)t @RT(0) @T @F @DT @RT(4)REAL @RT(0) @T @T @BASIC 0 @F
@F @F
@T
@BEG_Attrib
3 @RT(3)0.2 @RT(0) @RT(0)
@END_Attrib
1 0 @F @F @F @F

@Var @RT(1)T @RT(0) @T @F @DT @RT(4)REAL @RT(0) @T @T @BASIC 0 @F
@F @F
@T
@BEG_Attrib
3 @RT(0) @RT(0) @RT(0)
@END_Attrib
1 0 @F @F @F @F

@Var @RT(2)Kp @RT(0) @T @F @DT @RT(4)REAL @RT(0) @T @T @BASIC 0 @F
@F @F
@T
@BEG_Attrib
3 @RT(4)0.05 @RT(0) @RT(0)
@END_Attrib
1 0 @F @F @F @F

@Var @RT(2)Ti @RT(0) @T @F @DT @RT(4)REAL @RT(0) @T @T @BASIC 0 @F
@F @F
@T
@BEG_Attrib
3 @RT(0) @RT(0) @RT(0)
@END_Attrib
1 0 @F @F @F @F

@Var @RT(2)ti @RT(0) @T @F @DT @RT(4)REAL @RT(0) @T @T @BASIC 0 @F
@F @F
@T
@BEG_Attrib
3 @RT(4)0.05 @RT(0) @RT(0)
@END_Attrib
1 0 @F @F @F @F

@Var @RT(2)Td @RT(0) @T @F @DT @RT(4)REAL @RT(0) @T @T @BASIC 0 @F
@F @F
@T
@BEG_Attrib
3 @RT(0) @RT(0) @RT(0)
@END_Attrib
1 0 @F @F @F @F

@Var @RT(2)td @RT(0) @T @F @DT @RT(4)REAL @RT(0) @T @T @BASIC 0 @F
@F @F
@T
@BEG_Attrib
3 @RT(3)2.0 @RT(0) @RT(0)
@END_Attrib
1 0 @F @F @F @F

@Var @RT(1)A @RT(0) @T @F @DT @RT(4)REAL @RT(0) @T @T @BASIC 0 @F
@F @F
@T
@BEG_Attrib
3 @RT(0) @RT(0) @RT(0)
@END_Attrib
1 0 @F @F @F @F

@Var @RT(1)B @RT(0) @T @F @DT @RT(4)REAL @RT(0) @T @T @BASIC 0 @F
@F @F
@T
@BEG_Attrib
3 @RT(0) @RT(0) @RT(0)
@END_Attrib
1 0 @F @F @F @F

@Var @RT(1)C @RT(0) @T @F @DT @RT(4)REAL @RT(0) @T @T @BASIC 0 @F
@F @F
@T
@BEG_Attrib
3 @RT(0) @RT(0) @RT(0)
@END_Attrib
1 0 @F @F @F @F

@Var @RT(12)di_ButtonBwd @RT(0) @T @F @DT @RT(4)BOOL @RT(0) @T @T @BASIC 0 @F
@F @F
@T
@BEG_Attrib
3 @RT(0) @RT(11)Panelbutton @RT(0)
@END_Attrib
1 8 @F @F @F @F

@Var @RT(12)di_ButtonFwd @RT(0) @T @F @DT @RT(4)BOOL @RT(0) @T @T @BASIC 0 @F
@F @F
@T
@BEG_Attrib
3 @RT(0) @RT(11)Panelbutton @RT(0)
@END_Attrib
1 8 @F @F @F @F

@Var @RT(6)ao_pid @RT(0) @T @F @DT @RT(4)REAL @RT(0) @T @T @BASIC 0 @F
@F @F
@T
@BEG_Attrib
3 @RT(0) @RT(0) @RT(0)
@END_Attrib
1 8 @F @F @F @F

@Var @RT(6)ai_pid @RT(0) @T @F @DT @RT(4)REAL @RT(0) @T @T @BASIC 0 @F
@F @F
@T
@BEG_Attrib
3 @RT(4)10.0 @RT(0) @RT(0)
@END_Attrib
1 0 @F @F @F @F

@Var @RT(9)PU_Task_7 @RT(0) @T @T @RENAMED 0 @T @T @DT @RT(4)TASK @RT(0) @T @T @BASIC 0 @F
@F @F
@T
@BEG_Attrib
3 @RT(0) @RT(0) @RT(0)
@END_Attrib
1 7 @F @F @F @F

@Var @RT(9)PWMPeriod @RT(0) @T @F @DT @RT(4)TIME @RT(0) @T @T @BASIC 0 @F
@F @F
@T
@BEG_Attrib
3 @RT(0) @RT(0) @RT(0)
@END_Attrib
1 0 @F @F @F @F

@Var @RT(5)T_PID @RT(0) @T @F @DT @RT(4)REAL @RT(0) @T @T @BASIC 0 @F
@F @F
@T
@BEG_Attrib
3 @RT(0) @RT(0) @RT(0)
@END_Attrib
1 0 @F @F @F @F

@Var @RT(3)L_T @RT(0) @T @F @DT @RT(4)REAL @RT(0) @T @T @BASIC 0 @F
@F @F
@T
@BEG_Attrib
3 @RT(0) @RT(0) @RT(0)
@END_Attrib
1 0 @F @F @F @F

@Var @RT(3)H_T @RT(0) @T @F @DT @RT(4)REAL @RT(0) @T @T @BASIC 0 @F
@F @F
@T
@BEG_Attrib
3 @RT(0) @RT(0) @RT(0)
@END_Attrib
1 0 @F @F @F @F

@Var @RT(9)DutyRatio @RT(0) @T @F @DT @RT(4)REAL @RT(0) @T @T @BASIC 0 @F
@F @F
@T
@BEG_Attrib
3 @RT(0) @RT(0) @RT(0)
@END_Attrib
1 0 @F @F @F @F

@Var @RT(10)erCopyDone @RT(0) @T @F @DT @RT(5)ALARM @RT(0) @T @T @BASIC 0 @F
@F @T
@T
@BEG_Attrib
3 @RT(0) @RT(0) @RT(0)
@END_Attrib
1 7 @F @F @F @F

@Var @RT(12)sv_PathArray @RT(0) @T @T @DERIVED 0 @T @T @DT @RT(13)UsbFilesArray @RT(0) @T @T @UNKNOWN 0 @F
@F @F
@T
@BEG_Attrib
3 @RT(0) @RT(0) @RT(0)
@END_Attrib
1 8 @F @F @F @F

@Var @RT(14)sv_PathDisplay @RT(0) @T @T @DERIVED 0 @T @T @DT @RT(7)UsbFile @RT(0) @T @T @UNKNOWN 0 @F
@F @T
@T
@BEG_Attrib
3 @RT(0) @RT(0) @RT(0)
@END_Attrib
1 8 @F @F @F @F

@Var @RT(13)sv_rActOutput @RT(0) @T @F @DT @RT(3)INT @RT(0) @T @T @BASIC 0 @F
@F @F
@T
@BEG_Attrib
3 @RT(0) @RT(0) @RT(0)
@END_Attrib
1 8 @F @F @F @F

@Var @RT(13)sv_rSetOutput @RT(0) @T @F @DT @RT(3)INT @RT(0) @T @T @BASIC 0 @F
@F @F
@T
@BEG_Attrib
3 @RT(0) @RT(0) @RT(0)
@END_Attrib
1 8 @F @F @F @F

@Var @RT(12)sv_bStartPID @RT(0) @T @F @DT @RT(4)BOOL @RT(0) @T @T @BASIC 0 @F
@F @F
@T
@BEG_Attrib
3 @RT(0) @RT(0) @RT(0)
@END_Attrib
1 8 @F @F @F @F

@Var @RT(19)fbReadIOConfigFiles @RT(0) @T @T @DERIVED 0 @T @T @DT @RT(19)FBReadIOConfigFiles @RT(0) @T @T @UNKNOWN 0 @F
@F @F
@T
@BEG_Attrib
3 @RT(0) @RT(0) @RT(0)
@END_Attrib
1 0 @F @F @F @F

@END_Dcl

@END_Export

@BEG_Body

10

@BEG_Export

@BEG_Algo
@PROCESS_ALGORITHM @RT(22)paInitDebugMeasurement @STRUCTURED_TEXT
@RT(0) @RT(0) @RT(8)TaskSlow @T @F
@END_Algo

@BEG_Dcl
@RT(16)DclTreeContainer
4
@Var @RT(6)fuName @RT(0) @T @F @DT @RT(11)STRING(255) @RT(0) @T @T @STRING 0 @F @RT(3)255 @F
@F @F
@T
@BEG_Attrib
3 @RT(0) @RT(0) @RT(0)
@END_Attrib
1 0 @F @F @F @F

@Var @RT(12)variableName @RT(0) @T @F @DT @RT(11)STRING(255) @RT(0) @T @T @STRING 0 @F @RT(3)255 @F
@F @F
@T
@BEG_Attrib
3 @RT(0) @RT(0) @RT(0)
@END_Attrib
1 0 @F @F @F @F

@Var @RT(8)swoState @RT(0) @T @T @DERIVED 0 @T @T @DT @RT(11)KSWO_Status @RT(0) @T @T @UNKNOWN 0 @F
@F @F
@T
@BEG_Attrib
3 @RT(0) @RT(0) @RT(0)
@END_Attrib
1 0 @F @F @F @F

@Var @RT(1)b @RT(0) @T @F @DT @RT(4)BOOL @RT(0) @T @T @BASIC 0 @F
@F @F
@T
@BEG_Attrib
3 @RT(0) @RT(0) @RT(0)
@END_Attrib
1 0 @F @F @F @F

@END_Dcl

@END_Export

@BEG_Export

@BEG_Algo
@PROCESS_ALGORITHM @RT(9)paMeasure @SEQUENTIAL_FLOW_CHART
@RT(0) @RT(0) @RT(10)TaskAnalog @T @F
@END_Algo

@BEG_Dcl
@RT(16)DclTreeContainer
2
@Var @RT(16)abEjectorMeasure @RT(0) @T @T @DERIVED 0 @T @T @DT @RT(11)ABMeasureAI @RT(0) @T @T @UNKNOWN 0 @F
@F @F
@T
@BEG_Attrib
3 @RT(0) @RT(0) @RT(0)
@END_Attrib
1 0 @F @F @F @F

@Var @RT(1)b @RT(0) @T @F @DT @RT(4)BOOL @RT(0) @T @T @BASIC 0 @F
@F @F
@T
@BEG_Attrib
3 @RT(0) @RT(0) @RT(0)
@END_Attrib
1 4 @F @F @F @F

@END_Dcl

@END_Export

@BEG_Export

@BEG_Algo
@PROCESS_ALGORITHM @RT(5)paPID @SEQUENTIAL_FLOW_CHART
@RT(0) @RT(0) @RT(10)TaskAnalog @F @F
@END_Algo

@BEG_Dcl
@RT(16)DclTreeContainer
0
@END_Dcl

@END_Export

@BEG_Export

@BEG_Algo
@POSTUPDATE_ALGORITHM @RT(1)p @STRUCTURED_TEXT
@RT(0) @RT(25)di_ButtonBwd,di_ButtonFwd @RT(9)PU_Task_7 @F @F
@END_Algo

@BEG_Dcl
@RT(16)DclTreeContainer
1
@Var @RT(1)a @RT(0) @T @F @DT @RT(3)INT @RT(0) @T @T @BASIC 0 @F
@F @F
@T
@BEG_Attrib
3 @RT(0) @RT(0) @RT(0)
@END_Attrib
1 0 @F @F @F @F

@END_Dcl

@END_Export

@BEG_Export

@BEG_Algo
@PROCESS_ALGORITHM @RT(5)paPWM @SEQUENTIAL_FLOW_CHART
@RT(0) @RT(0) @RT(10)TaskAnalog @F @F
@END_Algo

@BEG_Dcl
@RT(16)DclTreeContainer
2
@Var @RT(5)fbTON @RT(0) @T @T @DERIVED 0 @T @T @DT @RT(3)TON @RT(0) @T @T @UNKNOWN 0 @F
@F @F
@T
@BEG_Attrib
3 @RT(0) @RT(0) @RT(0)
@END_Attrib
1 0 @F @F @F @F

@Var @RT(2)do @RT(0) @T @F @DT @RT(4)BOOL @RT(0) @T @T @BASIC 0 @F
@F @F
@T
@BEG_Attrib
3 @RT(0) @RT(0) @RT(0)
@END_Attrib
1 0 @F @F @F @F

@END_Dcl

@END_Export

@BEG_Export

@BEG_Algo
@POSTUPDATE_ALGORITHM @RT(3)USB @STRUCTURED_TEXT
@RT(0) @RT(25)di_ButtonBwd,di_ButtonFwd @RT(9)PU_Task_7 @F @F
@END_Algo

@BEG_Dcl
@RT(16)DclTreeContainer
1
@Var @RT(8)PLCFiles @RT(0) @T @F @DT @RT(11)STRING(255) @RT(0) @T @T @STRING 0 @F @RT(3)255 @F
@F @F
@T
@BEG_Attrib
3 @RT(18)'/harddisk0/PLCIO' @RT(0) @RT(0)
@END_Attrib
1 0 @F @F @F @F

@END_Dcl

@END_Export

@BEG_Export

@BEG_Algo
@PROCESS_ALGORITHM @RT(5)paUSB @SEQUENTIAL_FLOW_CHART
@RT(0) @RT(0) @RT(10)TaskAnalog @F @F
@END_Algo

@BEG_Dcl
@RT(16)DclTreeContainer
14
@Var @RT(11)Stable_Free @RT(0) @T @T @DERIVED 0 @T @T @DT @RT(12)KFILE_Status @RT(0) @T @T @UNKNOWN 0 @F
@F @F
@T
@BEG_Attrib
3 @RT(0) @RT(0) @RT(0)
@END_Attrib
1 0 @F @F @F @F

@Var @RT(13)Stable_Delete @RT(0) @T @T @DERIVED 0 @T @T @DT @RT(12)KFILE_Status @RT(0) @T @T @UNKNOWN 0 @F
@F @F
@T
@BEG_Attrib
3 @RT(0) @RT(0) @RT(0)
@END_Attrib
1 0 @F @F @F @F

@Var @RT(11)Stable_Copy @RT(0) @T @T @DERIVED 0 @T @T @DT @RT(12)KFILE_Status @RT(0) @T @T @UNKNOWN 0 @F
@F @F
@T
@BEG_Attrib
3 @RT(0) @RT(0) @RT(0)
@END_Attrib
1 0 @F @F @F @F

@Var @RT(11)Stable_Next @RT(0) @T @T @DERIVED 0 @T @T @DT @RT(12)KFILE_Status @RT(0) @T @T @UNKNOWN 0 @F
@F @F
@T
@BEG_Attrib
3 @RT(0) @RT(0) @RT(0)
@END_Attrib
1 0 @F @F @F @F

@Var @RT(12)Stable_First @RT(0) @T @T @DERIVED 0 @T @T @DT @RT(12)KFILE_Status @RT(0) @T @T @UNKNOWN 0 @F
@F @F
@T
@BEG_Attrib
3 @RT(0) @RT(0) @RT(0)
@END_Attrib
1 0 @F @F @F @F

@Var @RT(12)Stable_Copy2 @RT(0) @T @T @DERIVED 0 @T @T @DT @RT(12)KFILE_Status @RT(0) @T @T @UNKNOWN 0 @F
@F @F
@T
@BEG_Attrib
3 @RT(0) @RT(0) @RT(0)
@END_Attrib
1 0 @F @F @F @F

@Var @RT(13)Stable_Rename @RT(0) @T @T @DERIVED 0 @T @T @DT @RT(12)KFILE_Status @RT(0) @T @T @UNKNOWN 0 @F
@F @F
@T
@BEG_Attrib
3 @RT(0) @RT(0) @RT(0)
@END_Attrib
1 0 @F @F @F @F

@Var @RT(1)i @RT(0) @T @F @DT @RT(4)LINT @RT(0) @T @T @BASIC 0 @F
@F @F
@T
@BEG_Attrib
3 @RT(0) @RT(0) @RT(0)
@END_Attrib
1 0 @F @F @F @F

@Var @RT(10)SystemPath @RT(0) @T @F @DT @RT(11)STRING(255) @RT(0) @T @T @STRING 0 @F @RT(3)255 @F
@F @F
@T
@BEG_Attrib
3 @RT(77)'/harddisk0/application/control/config/KeStudio_generated/Device1/PlcIo.cfgr' @RT(0) @RT(0)
@END_Attrib
1 0 @F @F @F @F

@Var @RT(1)s @RT(0) @T @F @DT @RT(11)STRING(255) @RT(0) @T @T @STRING 0 @F @RT(3)255 @F
@F @F
@T
@BEG_Attrib
3 @RT(0) @RT(0) @RT(0)
@END_Attrib
1 0 @F @F @F @F

@Var @RT(2)s2 @RT(0) @T @F @DT @RT(11)STRING(255) @RT(0) @T @T @STRING 0 @F @RT(3)255 @F
@F @F
@T
@BEG_Attrib
3 @RT(0) @RT(0) @RT(0)
@END_Attrib
1 0 @F @F @F @F

@Var @RT(1)j @RT(0) @T @F @DT @RT(4)DINT @RT(0) @T @T @BASIC 0 @F
@F @F
@T
@BEG_Attrib
3 @RT(0) @RT(0) @RT(0)
@END_Attrib
1 4 @F @F @F @F

@Var @RT(9)harddisk0 @RT(0) @T @F @DT @RT(11)STRING(255) @RT(0) @T @T @STRING 0 @F @RT(3)255 @F
@F @F
@T
@BEG_Attrib
3 @RT(12)'/harddisk0' @RT(0) @RT(0)
@END_Attrib
1 0 @F @F @F @F

@Var @RT(8)PLCFiles @RT(0) @T @F @DT @RT(11)STRING(255) @RT(0) @T @T @STRING 0 @F @RT(3)255 @F
@F @F
@T
@BEG_Attrib
3 @RT(12)'/harddisk0' @RT(0) @RT(0)
@END_Attrib
1 0 @F @F @F @F

@END_Dcl

@END_Export

@BEG_Export

@BEG_Algo
@POSTUPDATE_ALGORITHM @RT(7)pchoose @STRUCTURED_TEXT
@RT(0) @RT(90)sv_bUse1,sv_bUse2,sv_bUse3,sv_bUse4,sv_bUse5,sv_bUse6,sv_bUse7,sv_bUse8,sv_bUse9,sv_bUse10 @RT(9)PU_Task_7 @F @T
@END_Algo

@BEG_Dcl
@RT(16)DclTreeContainer
2
@Var @RT(11)Stable_Copy @RT(0) @T @T @DERIVED 0 @T @T @DT @RT(12)KFILE_Status @RT(0) @T @T @UNKNOWN 0 @F
@F @F
@T
@BEG_Attrib
3 @RT(0) @RT(0) @RT(0)
@END_Attrib
1 0 @F @F @F @F

@Var @RT(10)SystemPath @RT(0) @T @F @DT @RT(11)STRING(255) @RT(0) @T @T @STRING 0 @F @RT(3)255 @F
@F @F
@T
@BEG_Attrib
3 @RT(77)'/harddisk0/application/control/config/KeStudio_generated/Device1/PlcIo.cfgr' @RT(0) @RT(0)
@END_Attrib
1 0 @F @F @F @F

@END_Dcl

@END_Export

@BEG_Export

@BEG_Algo
@PROCESS_ALGORITHM @RT(9)paPIDCalc @STRUCTURED_TEXT
@RT(0) @RT(0) @RT(10)TaskAnalog @T @T
@END_Algo

@BEG_Dcl
@RT(16)DclTreeContainer
0
@END_Dcl

@END_Export

@BEG_Export

@BEG_Algo
@PROCESS_ALGORITHM @RT(10)pStaratPID @STRUCTURED_TEXT
@RT(0) @RT(0) @RT(8)TaskSlow @T @F
@END_Algo

@BEG_Dcl
@RT(16)DclTreeContainer
6
@Var @RT(3)iKp @RT(0) @T @F @DT @RT(3)INT @RT(0) @T @T @BASIC 0 @F
@F @F
@T
@BEG_Attrib
3 @RT(1)2 @RT(0) @RT(0)
@END_Attrib
1 0 @F @F @F @F

@Var @RT(3)iKd @RT(0) @T @F @DT @RT(3)INT @RT(0) @T @T @BASIC 0 @F
@F @F
@T
@BEG_Attrib
3 @RT(1)1 @RT(0) @RT(0)
@END_Attrib
1 0 @F @F @F @F

@Var @RT(3)iKi @RT(0) @T @F @DT @RT(3)INT @RT(0) @T @T @BASIC 0 @F
@F @F
@T
@BEG_Attrib
3 @RT(1)1 @RT(0) @RT(0)
@END_Attrib
1 0 @F @F @F @F

@Var @RT(7)iFilter @RT(0) @T @F @DT @RT(3)INT @RT(0) @T @T @BASIC 0 @F
@F @F
@T
@BEG_Attrib
3 @RT(4)1023 @RT(0) @RT(0)
@END_Attrib
1 0 @F @F @F @F

@Var @RT(7)iIntegr @RT(0) @T @F @DT @RT(3)INT @RT(0) @T @T @BASIC 0 @F
@F @F
@T
@BEG_Attrib
3 @RT(1)0 @RT(0) @RT(0)
@END_Attrib
1 0 @F @F @F @F

@Var @RT(5)abPID @RT(0) @T @T @DERIVED 0 @F @RT(5)ABPID @F
@T
@BEG_Attrib
3 @RT(0) @RT(0) @RT(0)
@END_Attrib
1 0 @F @F @F @F

@END_Dcl

@END_Export

@BEG_Body
@TL(77)
fuName := GET_MY_FU_NAME();
variableName := CONCAT(fuName,'.rPosition mm');
swoState := KSWO_AddVariable( Task := TaskAnalog,
                              Name := variableName,
                              Variable := sv_rEjectorPosition);
b := FAddToScopeGroup(Task := TaskAnalog,
                      Name := variableName,
                      GroupId := cScopeGroupEjector);
variableName := CONCAT(fuName,'.rVelocity mm/s');
swoState := KSWO_AddVariable( Task := TaskAnalog,
                              Name := variableName,
                              Variable := sv_rEjectorVelocity);
b := FAddToScopeGroup(Task := TaskAnalog,
                      Name := variableName,
                      GroupId := cScopeGroupEjector);

    variableName := CONCAT(fuName,'.sv_Ek');
swoState := KSWO_AddVariable( Task := TaskAnalog,
                              Name := variableName,
                              Variable := sv_Ek);

    variableName := CONCAT(fuName,'.sv_Uk');
swoState := KSWO_AddVariable( Task := TaskAnalog,
                              Name := variableName,
                              Variable := sv_Uk);

    variableName := CONCAT(fuName,'.sv_Ui');
swoState := KSWO_AddVariable( Task := TaskAnalog,
                              Name := variableName,
                              Variable := sv_Ui);

    variableName := CONCAT(fuName,'.ao_pid');
swoState := KSWO_AddVariable( Task := TaskAnalog,
                              Name := variableName,
                              Variable := ao_pid);

    variableName := CONCAT(fuName,'.ai_pid');
swoState := KSWO_AddVariable( Task := TaskAnalog,
                              Name := variableName,
                              Variable := ai_pid);

    variableName := CONCAT(fuName,'.sv_rActOutput');
swoState := KSWO_AddVariable( Task := TaskAnalog,
                              Name := variableName,
                              Variable := sv_rActOutput);
    variableName := CONCAT(fuName,'.sv_rSetOutput');
swoState := KSWO_AddVariable( Task := TaskAnalog,
                              Name := variableName,
                              Variable := sv_rSetOutput);

STOP_PROCESS_ALGORITHM();

@END_Body

@@@BEG_Comment@@@
@TL(0)

@@@END_Comment@@@

@BEG_SfcBody
4 6 5

@BEG_SfcData 2
@StepSeq @RT(4)sseq @F 5
@Step @RT(7)S_Start @F @T @T @F @RT(0) @F
@AcbCont @RT(7)unnamed @F 0

@AltBranch @RT(3)alt @F 2
@TransSeq @RT(4)tseq @F 1
@Trans @RT(7)TLinked @F @T @F @F @T @T @TL(2)
IS_LINKED(ai_Position)

@RT(7)TLinked @F

@TransSeq @RT(4)tseq @F 4
@Trans @RT(10)TNotLinked @F @T @F @F @T @T @TL(2)
NOT IS_LINKED(ai_Position)

@RT(10)TNotLinked @F
@Step @RT(6)S_Stop @F @F @F @F @RT(0) @F
@AcbCont @RT(7)unnamed @F 1
@Acb @RT(5)AStop @F @T @RT(1)P @RT(0) @F @F @T @TL(2)
STOP_PROCESS_ALGORITHM();

@F

@Trans @RT(5)TStop @F @T @F @F @T @T @TL(2)
TRUE

@RT(5)TStop @F
@Goto @RT(7)S_Start @F @F

@Step @RT(6)S_Init @F @F @F @F @RT(0) @F
@AcbCont @RT(7)unnamed @F 1
@Acb @RT(17)AInitMeasureBlock @F @F @RT(1)P @RT(0) @F @F @F @F

@Trans @RT(9)TInitDone @F @T @F @F @T @T @TL(2)
TRUE

@RT(9)TInitDone @F
@Step @RT(9)S_Measure @F @F @F @F @RT(0) @F
@AcbCont @RT(7)unnamed @F 1
@Acb @RT(8)AMeasure @F @F @RT(1)N @RT(0) @F @F @F @F

@END_SfcData
@SaActions 2
@SaText @RT(8)AMeasure 1 @TL(6)

abEjectorMeasure.aRun(bIdle := sv_bDeviceReady);
sv_bTransducerError := abEjectorMeasure.aRun.bSensorError;
b := WRITE_SVREAL_DIRECT(sv_rEjectorPosition, abEjectorMeasure.aRun.rValue);
b := WRITE_SVREAL_DIRECT(sv_rEjectorVelocity, abEjectorMeasure.aRun.rVelocity);

@SaText @RT(17)AInitMeasureBlock 1 @TL(9)

abEjectorMeasure.aInit(sRawValue := 'Ejector1.ai_Position',
                        pLintab := @sv_EjectorLintab);

abEjectorMeasure.aInitMonitoring(bEnable := sv_EjectorMonitorMeas.EnableMonitoring,
                                 rLowLimit := sv_EjectorMonitorMeas.LowerLimit,
                                 bLimitation := sv_EjectorMonitorMeas.Limitation,
                                 rFailureFactor := sv_EjectorMonitorMeas.FailureFactor);

@SaTrans 0
@SaExits 0
@END_SfcBody

@@@BEG_Comment@@@
@TL(0)

@@@END_Comment@@@

@BEG_SfcBody
5 5 6

@BEG_SfcData 2
@StepSeq @RT(4)sseq @F 5
@Step @RT(5)Step1 @F @T @F @F @RT(0) @F
@AcbCont @RT(7)unnamed @F 1
@Acb @RT(9)Action223 @F @T @RT(1)P @RT(0) @F @F @T @TL(6)
ai_pid := 10.0;
t := 0.1;
td := 2.0;
ti := 0.05;
Kp := 0.2;

@F

@Trans @RT(6)Trans1 @F @T @F @F @T @F @TL(2)
TRUE

@RT(6)Trans1 @F
@Step @RT(5)Step2 @F @F @F @F @RT(0) @F
@AcbCont @RT(7)unnamed @F 1
@Acb @RT(7)Action2 @F @T @RT(1)P @RT(0) @F @F @T @TL(10)
sv_Ek := 0.0;
sv_Ek_1 := 0.0;
sv_Ek_2 := 0.0;
sv_Uk := 0.0;
sv_Uk_1 := 0.0;
sv_Uk_2 := 0.0;
sv_Uk_3 := 0.0;

@F

@Trans @RT(6)Trans4 @F @T @F @F @T @T @TL(2)
TRUE

@RT(6)Trans4 @F
@Loop @RT(4)loop @F 2
@StepSeq @RT(3)seq @F 3
@Step @RT(5)Step4 @F @F @F @F @RT(0) @F
@AcbCont @RT(7)unnamed @F 0

@Trans @RT(6)Trans2 @F @T @F @F @T @T @TL(2)
Step4.T > t#0.1s

@RT(6)Trans2 @F
@Step @RT(5)Step3 @F @F @F @F @RT(0) @F
@AcbCont @RT(7)unnamed @F 1
@Acb @RT(7)Action3 @F @T @RT(1)P @RT(0) @F @F @T @TL(18)
T := 1.0/t;
Td := 1.0/td;
Ti := 1.0/ti;
A := Kp*(1.0 + T/Ti + Td/T);
B := Kp*(1.0 + 2.0*Td/T);
C := Kp*Td/T;
sv_Uk_3 := sv_Uk_2;
sv_Uk_2 := sv_Uk_1;
sv_Uk_1 := sv_Uk;
sv_Ek_2 := sv_Ek_1;
sv_Ek_1 := sv_Ek;
sv_Ek := ai_pid - sv_Uk;
sv_Ui := A*sv_Ek + B*sv_Ek_1 + C*sv_Ek_2;
ao_pid := sv_Uk_1 + sv_Ui;
sv_Uk := sv_Uk_1 + sv_Ui;

@F

@Trans @RT(6)Trans5 @F @T @T @T @T @F @TL(2)
TRUE

@RT(6)Trans5 @F

@END_SfcData
@SaActions 0
@SaTrans 0
@SaExits 0
@END_SfcBody

@@@BEG_Comment@@@
@TL(0)

@@@END_Comment@@@

@BEG_Body
@TL(13)

IF di_ButtonFwd THEN
   START_PROCESS_ALGORITHM(paPID);
   START_PROCESS_ALGORITHM(paPWM);

END_IF;

IF di_ButtonBwd THEN
   STOP_PROCESS_ALGORITHM(paPID);
   STOP_PROCESS_ALGORITHM(paPWM);
END_IF;
//year=(year%100==0)?(year%400==0?1:0):(year%4==0?1:0)

@END_Body

@@@BEG_Comment@@@
@TL(0)

@@@END_Comment@@@

@BEG_SfcBody
8 7 13

@BEG_SfcData 2
@StepSeq @RT(4)sseq @F 3
@Step @RT(5)Step1 @F @T @F @F @RT(0) @F
@AcbCont @RT(7)unnamed @F 1
@Acb @RT(8)Action20 @F @T @RT(1)P @RT(0) @F @F @T @TL(2)
PWMPeriod := t#2s;

@F

@Trans @RT(6)Trans1 @F @T @F @F @T @T @TL(2)
TRUE

@RT(6)Trans1 @F
@Loop @RT(4)loop @F 2
@StepSeq @RT(3)seq @F 5
@Step @RT(5)Step2 @F @F @F @F @RT(0) @F
@AcbCont @RT(7)unnamed @F 1
@Acb @RT(7)Action2 @F @T @RT(1)P @RT(0) @F @F @T @TL(13)
T_PID := ao_pid;
L_T := 8.0;
H_T := 10.0;
IF T_PID < L_T THEN
   DutyRatio := 1.0;
ELSE IF T_PID >= H_T - 0.1 THEN
   DutyRatio := 0.0;
ELSE
   DutyRatio := (T_PID - L_T) /(H_T - L_T);
END_IF;
END_IF;
fbTON(IN := FALSE);

@F

@Trans @RT(6)Trans2 @F @T @F @F @T @T @TL(2)
TRUE

@RT(6)Trans2 @F
@Step @RT(5)Step5 @F @F @F @F @RT(0) @F
@AcbCont @RT(7)unnamed @F 1
@Acb @RT(7)Action3 @F @T @RT(1)N @RT(0) @F @F @T @TL(9)
fbTON(IN := TRUE,
     // PT := REAL_TO_TIME(TIME_TO_REAL(PWMPeriod) * DutyRatio);
            PT := PWMPeriod * DutyRatio);
IF fbTON.Q THEN
   do := FALSE;
ELSE
   do := TRUE;
END_IF;

@F

@Trans @RT(7)Trans11 @F @T @F @F @T @T @TL(2)
Step5.T > PWMPeriod

@RT(7)Trans11 @F
@Step @RT(5)Step3 @F @F @F @F @RT(0) @F
@AcbCont @RT(7)unnamed @F 0

@Trans @RT(7)Trans12 @F @T @T @T @T @T @TL(2)
TRUE

@RT(7)Trans12 @F

@END_SfcData
@SaActions 0
@SaTrans 0
@SaExits 0
@END_SfcBody

@@@BEG_Comment@@@
@TL(0)

@@@END_Comment@@@

@BEG_Body
@TL(7)
IF di_ButtonBwd THEN
   START_PROCESS_ALGORITHM(paUSB);
END_IF;
IF di_ButtonFwd THEN
   STOP_PROCESS_ALGORITHM(paUSB);
END_IF;

@END_Body

@@@BEG_Comment@@@
@TL(0)

@@@END_Comment@@@

@BEG_SfcBody
7 7 7

@BEG_SfcData 2
@StepSeq @RT(4)sseq @F 1
@Loop @RT(4)loop @F 2
@StepSeq @RT(3)seq @F 5
@Step @RT(5)Step1 @F @T @F @F @RT(0) @F
@AcbCont @RT(7)unnamed @F 1
@Acb @RT(7)Action1 @F @T @RT(1)P @RT(0) @F @F @T @TL(3)
//Check harddisk left memory
Stable_Free :=  KFILE_VolumeFree(harddisk0,i)

@F

@Trans @RT(6)Trans3 @F @T @F @F @T @T @TL(2)
Stable_Free = KFILE_Status_OK

@RT(6)Trans3 @F
@Step @RT(5)Step4 @F @F @F @F @RT(0) @F
@AcbCont @RT(7)unnamed @F 1
@Acb @RT(7)Action3 @F @T @RT(1)P @RT(0) @F @F @T @TL(11)
//get first file name in the file
Stable_First := KFILE_GetFirst(PLCFiles,s);
sv_PathArray[1] := s;
s2 := s;
FOR j :=2 TO 10 DO
   //get other file name in the file
   Stable_Next := KFILE_GetNext(s2,s2);
   sv_PathArray[j] := s2;
END_FOR;
//Now all file name in sv_PathArray

@F

@Trans @RT(6)Trans5 @F @T @F @F @T @T @TL(2)
Stable_Next = KFILE_Status_NOTOK

@RT(6)Trans5 @F
@Step @RT(5)Step2 @F @F @F @F @RT(0) @F
@AcbCont @RT(7)unnamed @F 1
@Acb @RT(7)Action5 @F @T @RT(1)N @RT(0) @F @F @T @TL(3)

STOP_PROCESS_ALGORITHM();

@F

@Trans @RT(6)Trans2 @F @T @T @T @T @T @TL(2)
TRUE

@RT(6)Trans2 @F

@END_SfcData
@SaActions 0
@SaTrans 0
@SaExits 0
@END_SfcBody

@@@BEG_Comment@@@
@TL(0)

@@@END_Comment@@@

@BEG_Body
@TL(41)
IF sv_bUse1 THEN
Stable_Copy := KFILE_Copy(sv_PathDisplay.plc1,SystemPath);
END_IF;

IF sv_bUse2 THEN
Stable_Copy := KFILE_Copy(sv_PathDisplay.plc2,SystemPath);
END_IF;

IF sv_bUse3  THEN
Stable_Copy := KFILE_Copy(sv_PathDisplay.plc3,SystemPath);
END_IF;

IF sv_bUse4 THEN
Stable_Copy := KFILE_Copy(sv_PathDisplay.plc4,SystemPath);
END_IF;

IF sv_bUse5 THEN
Stable_Copy := KFILE_Copy(sv_PathDisplay.plc5,SystemPath);
END_IF;

IF sv_bUse6 THEN
Stable_Copy := KFILE_Copy(sv_PathDisplay.plc6,SystemPath);
END_IF;

IF sv_bUse7 THEN
Stable_Copy := KFILE_Copy(sv_PathDisplay.plc7,SystemPath);
END_IF;

IF sv_bUse8 THEN
Stable_Copy := KFILE_Copy(sv_PathDisplay.plc8,SystemPath);
END_IF;

IF sv_bUse9 THEN
Stable_Copy := KFILE_Copy(sv_PathDisplay.plc9,SystemPath);
END_IF;

IF sv_bUse10 THEN
Stable_Copy := KFILE_Copy(sv_PathDisplay.plc10,SystemPath);
END_IF;

@END_Body

@@@BEG_Comment@@@
@TL(0)

@@@END_Comment@@@

@BEG_Body
@TL(15)
Td := 1.0/td;
Ti := 1.0/ti;
A := Kp*(1.0 + T/Ti + Td/T);
B := Kp*(1.0 + 2.0*Td/T);
C := Kp*Td/T;
sv_Uk_3 := sv_Uk_2;
sv_Uk_2 := sv_Uk_1;
sv_Uk_1 := sv_Uk;
sv_Ek_2 := sv_Ek_1;
sv_Ek_1 := sv_Ek;
sv_Ek := ai_pid - sv_Uk;
sv_Ui := A*sv_Ek + B*sv_Ek_1 + C*sv_Ek_2;
ao_pid := sv_Uk_1 + sv_Ui;
sv_Uk := sv_Uk_1 + sv_Ui;

@END_Body

@@@BEG_Comment@@@
@TL(0)

@@@END_Comment@@@

@BEG_Body
@TL(15)
IF sv_bStartPID THEN
    abPID.aPID(iAct := (sv_rActOutput * 32/ 100),
         iSet := (sv_rSetOutput * 32 / 100),
         iKp := iKp,
         iKi := iKi,
         iKd := iKd,
         iC0 := iFilter,
         iYlow := -32,
         iYup := 32,
         iIntegr := iIntegr,
         iY => sv_rActOutput);
   iIntegr := abPID.aPID.iIntegr;

END_IF;

@END_Body

@@@BEG_Comment@@@
@TL(0)

@@@END_Comment@@@
@END_Body

@END_Contents

(* ---- ABPID.pu ---- *)
IMPORT_OVER_LISTFILE
 KSWO_Status

END_IMPORT

ALGORITHM_BLOCK ABPID #DUMMY_EDIT_BLOCK

SYSTEM_OBJECT
 TaskSlow : TASK;
 TaskAnalog : TASK;
 PU_Task_7 : TASK;
END_OBJECT

// PROCESS_ALGORITHM paInitDebugMeasurement ON TaskSlow AUTOSTART

// VAR
 // fuName : STRING(255);
 // variableName : STRING(255);
 // swoState : KSWO_Status;
 // b : BOOL;
// END_VAR
// #BEGIN_EDIT_BLOCK
// variableName := CONCAT(fuName,'.ai_pid');
// swoState := KSWO_AddVariable( Task := TaskAnalog,
//                               Name := variableName,
//                               Variable := ai_pid);
//
//
//
//
//
//
//
//
//
//
//
//
//
//
// STOP_PROCESS_ALGORITHM();

// ;#END_EDIT_BLOCK END_ALGORITHM

ALGORITHM aPID

VAR_INPUT
 iAct : INT;
 iKp : INT;
 iKd : INT;
 iKi : INT;
 iSet : INT;
 iC0 : INT;
END_VAR

VAR_OUTPUT
 iY : INT;
END_VAR

VAR_INPUT
 iYlow : INT;
 iYup : INT;
END_VAR

VAR_OUTPUT
 iFilter : INT;
END_VAR

VAR_IN_OUT
 iIntegr : INT;
END_VAR

VAR
 iYlowTemp : INT;
 iYupTemp : INT;
 iDummy : INT;
 iTemp : INT;
END_VAR
#BEGIN_EDIT_BLOCK

// sample limit values
iYlowTemp := iYlow;
iYupTemp := iYup;

// check limits for validity
IF iYupTemp < iYlowTemp THEN
    iDummy := iYupTemp;
    iYupTemp := iYlowTemp;
    iYlowTemp := iDummy;
END_IF;

// calculate gradient
iTemp := (iAct - (iFilter)) * (1024 - iC0);

// calculate PT1 Filter
iFilter := iFilter + (iTemp);

// calculate new output
iTemp := (iSet - iAct) * iKp + (0 - iTemp ) * iKd + (iIntegr);
iTemp := iTemp ;

// limit output between iYlow and iYup
iY := LIMIT(MN := iYlowTemp,
            IN := (iTemp),
            MX := iYupTemp);

// "integrator" feed (PT1)
iIntegr := iIntegr + ((iY) -iIntegr ) * (iKi);

;#END_EDIT_BLOCK END_ALGORITHM

END_ALGORITHM_BLOCK

#END_OF_IEC_PART

@Puma @IecEditor 6 152 @Pou 25
@@@BEG_Comment@@@

@@@END_Comment@@@

@BEG_Contents

@BEG_Func
@RT(17)FuncTreeContainer
0
@END_Func

@BEG_Const
@RT(18)ConstTreeContainer
0
@END_Const

@BEG_Export

@BEG_Kind
@ALGORITHM_BLOCK @RT(5)ABPID @STRUCTURED_TEXT
@RT(0) @RT(0) @RT(0)
@END_Kind

@BEG_Dcl
@RT(16)DclTreeContainer
3
@Var @RT(8)TaskSlow @RT(0) @T @F @DT @RT(4)TASK @RT(0) @T @T @BASIC 0 @F
@F @F
@T
@BEG_Attrib
3 @RT(0) @RT(0) @RT(0)
@END_Attrib
1 7 @F @F @F @F

@Var @RT(10)TaskAnalog @RT(0) @T @F @DT @RT(4)TASK @RT(0) @T @T @BASIC 0 @F
@F @F
@T
@BEG_Attrib
3 @RT(0) @RT(0) @RT(0)
@END_Attrib
1 7 @F @F @F @F

@Var @RT(9)PU_Task_7 @RT(0) @T @F @DT @RT(4)TASK @RT(0) @T @T @BASIC 0 @F
@F @F
@T
@BEG_Attrib
3 @RT(0) @RT(0) @RT(0)
@END_Attrib
1 7 @F @F @F @F

@END_Dcl

@END_Export

@BEG_Body

2

@BEG_Export

@BEG_Algo
@PROCESS_ALGORITHM @RT(22)paInitDebugMeasurement @STRUCTURED_TEXT
@RT(0) @RT(0) @RT(8)TaskSlow @T @T
@END_Algo

@BEG_Dcl
@RT(16)DclTreeContainer
4
@Var @RT(6)fuName @RT(0) @T @F @DT @RT(11)STRING(255) @RT(0) @T @T @STRING 0 @F @RT(3)255 @F
@F @F
@T
@BEG_Attrib
3 @RT(0) @RT(0) @RT(0)
@END_Attrib
1 0 @F @F @F @F

@Var @RT(12)variableName @RT(0) @T @F @DT @RT(11)STRING(255) @RT(0) @T @T @STRING 0 @F @RT(3)255 @F
@F @F
@T
@BEG_Attrib
3 @RT(0) @RT(0) @RT(0)
@END_Attrib
1 0 @F @F @F @F

@Var @RT(8)swoState @RT(0) @T @T @DERIVED 0 @T @T @DT @RT(11)KSWO_Status @RT(0) @T @T @UNKNOWN 0 @F
@F @F
@T
@BEG_Attrib
3 @RT(0) @RT(0) @RT(0)
@END_Attrib
1 0 @F @F @F @F

@Var @RT(1)b @RT(0) @T @F @DT @RT(4)BOOL @RT(0) @T @T @BASIC 0 @F
@F @F
@T
@BEG_Attrib
3 @RT(0) @RT(0) @RT(0)
@END_Attrib
1 0 @F @F @F @F

@END_Dcl

@END_Export

@BEG_Export

@BEG_Algo
@ALGORITHM @RT(4)aPID @STRUCTURED_TEXT
@RT(0) @RT(0) @RT(0) @F @F
@END_Algo

@BEG_Dcl
@RT(16)DclTreeContainer
15
@Var @RT(9)iYlowTemp @RT(0) @T @F @DT @RT(3)INT @RT(0) @T @T @BASIC 0 @F
@F @F
@T
@BEG_Attrib
3 @RT(0) @RT(0) @RT(0)
@END_Attrib
1 0 @F @F @F @F

@Var @RT(8)iYupTemp @RT(0) @T @F @DT @RT(3)INT @RT(0) @T @T @BASIC 0 @F
@F @F
@T
@BEG_Attrib
3 @RT(0) @RT(0) @RT(0)
@END_Attrib
1 0 @F @F @F @F

@Var @RT(6)iDummy @RT(0) @T @F @DT @RT(3)INT @RT(0) @T @T @BASIC 0 @F
@F @F
@T
@BEG_Attrib
3 @RT(0) @RT(0) @RT(0)
@END_Attrib
1 0 @F @F @F @F

@Var @RT(5)iTemp @RT(0) @T @F @DT @RT(3)INT @RT(0) @T @T @BASIC 0 @F
@F @F
@T
@BEG_Attrib
3 @RT(0) @RT(0) @RT(0)
@END_Attrib
1 0 @F @F @F @F

@Var @RT(4)iAct @RT(0) @T @F @DT @RT(3)INT @RT(0) @T @T @BASIC 0 @F
@F @F
@T
@BEG_Attrib
3 @RT(0) @RT(0) @RT(0)
@END_Attrib
1 1 @F @F @F @F

@Var @RT(3)iKp @RT(0) @T @F @DT @RT(3)INT @RT(0) @T @T @BASIC 0 @F
@F @F
@T
@BEG_Attrib
3 @RT(0) @RT(0) @RT(0)
@END_Attrib
1 1 @F @F @F @F

@Var @RT(3)iKd @RT(0) @T @F @DT @RT(3)INT @RT(0) @T @T @BASIC 0 @F
@F @F
@T
@BEG_Attrib
3 @RT(0) @RT(0) @RT(0)
@END_Attrib
1 1 @F @F @F @F

@Var @RT(3)iKi @RT(0) @T @F @DT @RT(3)INT @RT(0) @T @T @BASIC 0 @F
@F @F
@T
@BEG_Attrib
3 @RT(0) @RT(0) @RT(0)
@END_Attrib
1 1 @F @F @F @F

@Var @RT(4)iSet @RT(0) @T @F @DT @RT(3)INT @RT(0) @T @T @BASIC 0 @F
@F @F
@T
@BEG_Attrib
3 @RT(0) @RT(0) @RT(0)
@END_Attrib
1 1 @F @F @F @F

@Var @RT(3)iC0 @RT(0) @T @F @DT @RT(3)INT @RT(0) @T @T @BASIC 0 @F
@F @F
@T
@BEG_Attrib
3 @RT(0) @RT(0) @RT(0)
@END_Attrib
1 1 @F @F @F @F

@Var @RT(2)iY @RT(0) @T @F @DT @RT(3)INT @RT(0) @T @T @BASIC 0 @F
@F @F
@T
@BEG_Attrib
3 @RT(0) @RT(0) @RT(0)
@END_Attrib
1 3 @F @F @F @F

@Var @RT(5)iYlow @RT(0) @T @F @DT @RT(3)INT @RT(0) @T @T @BASIC 0 @F
@F @F
@T
@BEG_Attrib
3 @RT(0) @RT(0) @RT(0)
@END_Attrib
1 1 @F @F @F @F

@Var @RT(4)iYup @RT(0) @T @F @DT @RT(3)INT @RT(0) @T @T @BASIC 0 @F
@F @F
@T
@BEG_Attrib
3 @RT(0) @RT(0) @RT(0)
@END_Attrib
1 1 @F @F @F @F

@Var @RT(7)iFilter @RT(0) @T @F @DT @RT(3)INT @RT(0) @T @T @BASIC 0 @F
@F @F
@T
@BEG_Attrib
3 @RT(0) @RT(0) @RT(0)
@END_Attrib
1 3 @F @F @F @F

@Var @RT(7)iIntegr @RT(0) @T @F @DT @RT(3)INT @RT(0) @T @T @BASIC 0 @F
@F @F
@T
@BEG_Attrib
3 @RT(0) @RT(0) @RT(0)
@END_Attrib
1 2 @F @F @F @F

@END_Dcl

@END_Export

@BEG_Body
@TL(20)
variableName := CONCAT(fuName,'.ai_pid');
swoState := KSWO_AddVariable( Task := TaskAnalog,
                              Name := variableName,
                              Variable := ai_pid);

STOP_PROCESS_ALGORITHM();

@END_Body

@@@BEG_Comment@@@
@TL(0)

@@@END_Comment@@@

@BEG_Body
@TL(30)

// sample limit values
iYlowTemp := iYlow;
iYupTemp := iYup;

// check limits for validity
IF iYupTemp < iYlowTemp THEN
    iDummy := iYupTemp;
    iYupTemp := iYlowTemp;
    iYlowTemp := iDummy;
END_IF;

// calculate gradient
iTemp := (iAct - (iFilter)) * (1024 - iC0);

// calculate PT1 Filter
iFilter := iFilter + (iTemp);

// calculate new output
iTemp := (iSet - iAct) * iKp + (0 - iTemp ) * iKd + (iIntegr);
iTemp := iTemp ;

// limit output between iYlow and iYup
iY := LIMIT(MN := iYlowTemp,
            IN := (iTemp),
            MX := iYupTemp);

// "integrator" feed (PT1)
iIntegr := iIntegr + ((iY) -iIntegr ) * (iKi);

@END_Body

@@@BEG_Comment@@@
@TL(0)

@@@END_Comment@@@
@END_Body

@END_Contents
